Omron CX-Programmer project NewProject (CX-Programmer 9.73)

# PLC NewPLC1: CP1E N30

## Program NewProgram1 (cyclic task 0)
Local symbols
TR BOOL

### Section Section1

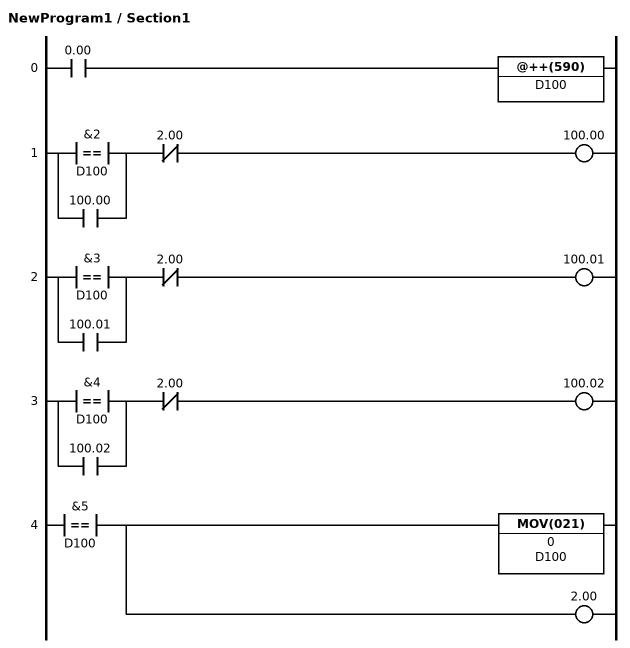
; rung 0
LD 0.00
@++(590) D100
; rung 1
LD=(300) &2 D100
OR 100.00
ANDNOT 2.00
OUT 100.00
; rung 2
LD=(300) &3 D100
OR 100.01
ANDNOT 2.00
OUT 100.01
; rung 3
LD=(300) &4 D100
OR 100.02
ANDNOT 2.00
OUT 100.02
; rung 4
LD=(300) &5 D100
MOV(021) 0 D100
OUT 2.00

### Section END
; rung 0
END(001)